INTERFACE I_SessionHeaderAccessor

METHOD PUBLIC TryGetSessionIdFromRequest : BOOL
VAR_INPUT
	Request : I_Request;
	Destination : REFERENCE TO T_MAXSTRING;
END_VAR
END_METHOD

METHOD PUBLIC UpdateRequestWithSessionId
VAR_INPUT
	Request : I_Request;
	SessionId : T_MAXSTRING;
END_VAR
END_METHOD

METHOD PUBLIC UpdateResponseWithSessionId
VAR_INPUT
	Response : I_ServerResponse;
	SessionId : T_MAXSTRING;
END_VAR
END_METHOD

END_INTERFACE

(* stored: Version 1.1.0.1, ProductVersion 3.1.4024.12
   Itf I_SessionHeaderAccessor: Id {eb3f87de-5aa8-44de-b748-33564e049b3c}
   Method TryGetSessionIdFromRequest: Id {75eab0e8-3ede-4f43-952c-fb2d1910a92b}
   Method UpdateRequestWithSessionId: Id {1c2fb640-ceac-4ec3-a97c-4a617193ae6a}
   Method UpdateResponseWithSessionId: Id {fff2909b-f691-4212-a025-6cafadf2f40b} *)
